	FUNCTION_BLOCK FB 343
	TITLE =G243M COUPLING DEVICE TURNER GERM 8
	//COPYRIGHT:    (C) 2009  BUHLER AG, CH-9240 UZWIL, SWITZERLAND
	//
	//PRODUCT:      WinCoS_BIW01_09
	//
	//TITLE:        COUPLING DEVICE TURNER GERM 8
	//                Machine group control
	//                Maschinengruppensteuerung
	//
	//--------------------------------------------------------------------------------
	//
	//IDENT:        AUTHOR:             DEPT:                              DATE:
	//
	//P01_FB343.1.0 K.Renz              CSB41                              02.Apr.2010
	//             1st Release
	//
	//--------------------------------------------------------------------------------
	//
	//PURPOSE:
	//
	//MANUAL :
	//
	//RESTRICTIONS:
	//
	//--------------------------------------------------------------------------------
	AUTHOR  : KR
	FAMILY  : USW
	VERSION : 9.9


	VAR
	  Gr       : FB10;	//Standard interface to group
	  InOutValue1    : DINT; //Data for user
	  InOutValue2    : DINT; //Data for user
	  OutWayConflict : BOOL;	//Data for user
	  OutSelectionOk : BOOL;	//Data for user
	  CmdNewValue : BOOL;	//Data for user
	  CmdNewJob   : BOOL;	//Data for user
	  OutCodeOK   : BOOL;	//Data for user
	  InEndOfJob  : BOOL ;	//Data for user
	  staWayOk      : BOOL ;	//Data for user
	  EdgeStartRelease : BOOL ;	//Data for user
	  USW8  : BOOL;	//Data for user
	  USW9 : BOOL;	//Data for user
	  USW10: BOOL;	//Data for user
	  USW11: BOOL;	//Data for user
	  USW12: BOOL;	//Data for user
	  USW13: BOOL;	//Data for user
	  USW14: BOOL;	//Data for user
	  USW15: BOOL;	//Data for user
	     #A_2811_MXZ21 : FB12;   // Motor
	     #A_2811_BZS22 : FB14;   // DigInpCont
	     #A_2811_BZS23 : FB14;   // DigInpCont
	     #A_2811_MXZ25 : FB12;   // Motor
	     #A_2811_BZS26 : FB14;   // DigInpCont
	     #A_2811_BZS27 : FB14;   // DigInpCont
	     #A_2811_MXZ31 : FB12;   // Motor
	     #A_2811_BZS32 : FB14;   // DigInpCont
	     #A_2811_BZS33 : FB14;   // DigInpCont
	     #A_2811_MXZ35 : FB12;   // Motor
	     #A_2811_BZS37 : FB14;   // DigInpCont
	     #A_2811_BZS36 : FB14;   // DigInpCont
	END_VAR
	VAR_TEMP
	   tmpEnable		: BOOL;
	   tmpFlag  		: BOOL;
	   tmpCmdNext		: BOOL;
	   tmpLocal  		: BOOL;
	   tmpAspOk  		: BOOL;
	   tmpHWStop 		: BOOL;
	   tmpInstanzDBNo       : INT ;
	END_VAR
	BEGIN
	NETWORK
	TITLE =
	NETWORK
	TITLE =Read command from group control
	//Parameter
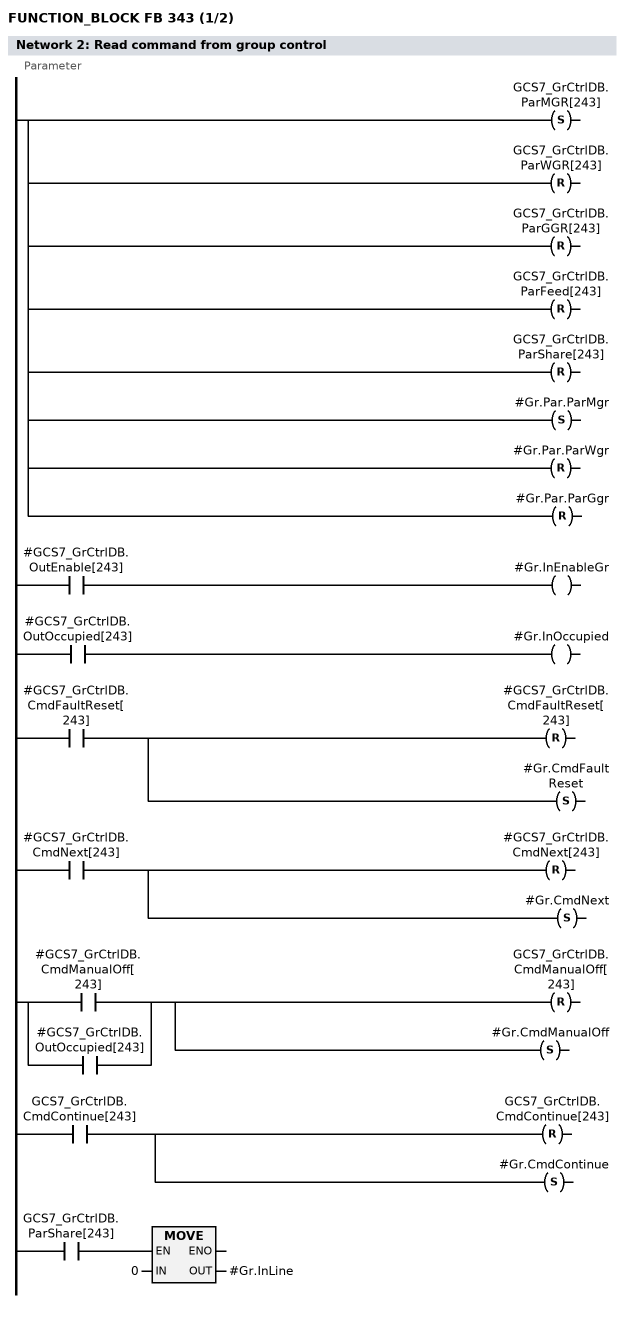
	      SET;
	      S   GCS7_GrCtrlDB.ParMGR[243];
	      R   GCS7_GrCtrlDB.ParWGR[243];
	      R   GCS7_GrCtrlDB.ParGGR[243];
	      R   GCS7_GrCtrlDB.ParFeed[243];
	      R   GCS7_GrCtrlDB.ParShare[243];
	      S   #Gr.Par.ParMgr;
	      R   #Gr.Par.ParWgr;
	      R   #Gr.Par.ParGgr;
	//Command
	      U   #GCS7_GrCtrlDB.OutEnable[243];
	      =   #Gr.InEnableGr;
	      U   #GCS7_GrCtrlDB.OutOccupied[243];
	      =   #Gr.InOccupied;
	      U   #GCS7_GrCtrlDB.CmdFaultReset[243];
	      R   #GCS7_GrCtrlDB.CmdFaultReset[243];
	      S   #Gr.CmdFaultReset;
	      U  #GCS7_GrCtrlDB.CmdNext[243];
	      R   #GCS7_GrCtrlDB.CmdNext[243];
	      S   #Gr.CmdNext;
	      U   #GCS7_GrCtrlDB.CmdManualOff[243];
	      O   #GCS7_GrCtrlDB.OutOccupied[243];
	      R   GCS7_GrCtrlDB.CmdManualOff[243];
	      S   #Gr.CmdManualOff;
	      U  GCS7_GrCtrlDB.CmdContinue[243];
	      R   GCS7_GrCtrlDB.CmdContinue[243];
	      S   #Gr.CmdContinue;
	//Init Line Number
	      U   GCS7_GrCtrlDB.ParShare[243];
	      SPBN WE00;
	      L     0;
	      T     #Gr.InLine;
	WE00: NOP   0;
	NETWORK
	TITLE =Call Methode Control
	// 1. Handle Interface PCControl
	// 2. Prepare mode --> ModePassive,ModeActive,ModeIdling
	// 3. Reset global flags of the group
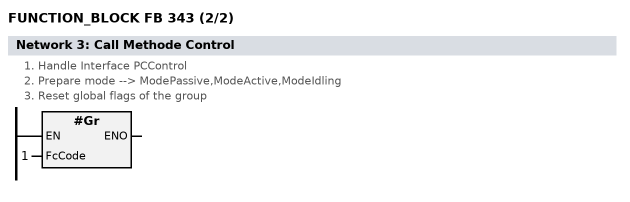
	      CALL #Gr (
	           FcCode                   := 1);
	NETWORK
	TITLE =Restart Idling Time
		L  #Gr.Par.ParIdling;
		L  2;
		>=I;
		SPB IdTm;
		T  #Gr.Par.ParIdling;
	IdTm:   NOP 0;
	      CLR;
	      S    #Gr.CmdRestartIdling;
	NETWORK
	TITLE =Prepare global flags
	NETWORK
	TITLE =Set Pattern (Target position)
	NETWORK
	TITLE =Interlocking WayOk
	//
	NETWORK
	TITLE =Interlocking Autostart
		CLR;
		R   #Gr.OutAutostart;
	NETWORK
	TITLE =Interlocking Enable
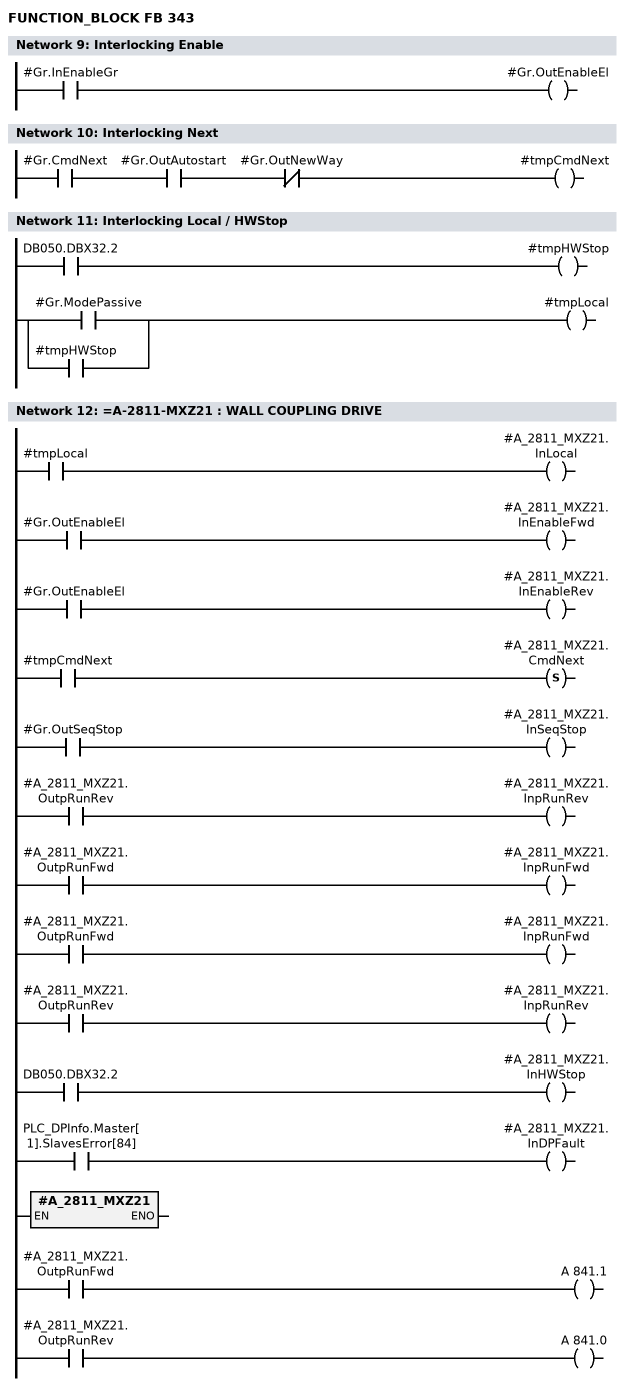
	      U     #Gr.InEnableGr;
	      =     #Gr.OutEnableEl;

	NETWORK
	TITLE =Interlocking Next
	      U     #Gr.CmdNext;
	      U     #Gr.OutAutostart;
	      UN    #Gr.OutNewWay;
	      =    #tmpCmdNext;

	NETWORK
	TITLE =Interlocking Local / HWStop
	      U    DB050.DBX32.2;
	      =    #tmpHWStop;

	      U    #Gr.ModePassive;
	      O    #tmpHWStop;
	      =    #tmpLocal;

	NETWORK
	TITLE ==A-2811-MXZ21 : WALL COUPLING DRIVE
	NOP 0;
	//-InLocal---
	      U     #tmpLocal;
	      =     #A_2811_MXZ21.InLocal;
	//
	//-Interlocking---
	      U     #Gr.OutEnableEl;
	      =     #A_2811_MXZ21.InEnableFwd;
	      U     #Gr.OutEnableEl;
	      =     #A_2811_MXZ21.InEnableRev;
	//
	      U    #tmpCmdNext;
	      S     #A_2811_MXZ21.CmdNext;
	//
	      U     #Gr.OutSeqStop;
	      =     #A_2811_MXZ21.InSeqStop;
	//
	//-Read inputs---
	      U     #A_2811_MXZ21.OutpRunRev;
	      =     #A_2811_MXZ21.InpRunRev;
	      U     #A_2811_MXZ21.OutpRunFwd;
	      =     #A_2811_MXZ21.InpRunFwd;
	      U     #A_2811_MXZ21.OutpRunFwd;
	      =     #A_2811_MXZ21.InpRunFwd;
	      U     #A_2811_MXZ21.OutpRunRev;
	      =     #A_2811_MXZ21.InpRunRev;
	      U   DB050.DBX32.2;
	      =     #A_2811_MXZ21.InHWStop;
	       U     PLC_DPInfo.Master[1].SlavesError[84];
	       =       #A_2811_MXZ21.InDPFault;
	//
	//-Set Parameters---
	//
	//-Call object control---
	      CALL  #A_2811_MXZ21;
	//
	//-Write outputs---
	      U     #A_2811_MXZ21.OutpRunFwd;
	      =     A 841.1;
	      U     #A_2811_MXZ21.OutpRunRev;
	      =     A 841.0;
	NETWORK
	TITLE ==A-2811-BZS22 : COUPLING DRIVE UNLOCKED
	NOP 0;
	//-InLocal---
	      U     #tmpLocal;
	      =     #A_2811_BZS22.InLocal;
	//
	//-Monitoring---
	      CLR;
	      =      #A_2811_BZS22.InMonTrue;
	      CLR;
	      =      #A_2811_BZS22.InMonFalse;
	//
	//-PreAlarm---
	      CLR;
	      =      #A_2811_BZS22.InPreAlarmTrue;
	      CLR;
	      =      #A_2811_BZS22.InPreAlarmFalse;
	//
	//-Additional commands---
	//      CLR
	//      S     #A_2811_BZS22.CmdRunTimeOutTime
	//
	//-Read inputs---
	      U     E 843.0;
	      =     #A_2811_BZS22.InpTrue;
	      U   DB050.DBX32.2;
	      =     #A_2811_BZS22.InHWStop;
	       U     PLC_DPInfo.Master[1].SlavesError[84];
	       =       #A_2811_BZS22.InDPFault;
	//
	//-Set Parameters---
	//
	//-Call object control---
	      CALL  #A_2811_BZS22;
	//
	//-Write outputs---
	NETWORK
	TITLE ==A-2811-BZS23 : COUPLING DRIVE LOCKED
	NOP 0;
	//-InLocal---
	      U     #tmpLocal;
	      =     #A_2811_BZS23.InLocal;
	//
	//-Monitoring---
	      CLR;
	      =      #A_2811_BZS23.InMonTrue;
	      CLR;
	      =      #A_2811_BZS23.InMonFalse;
	//
	//-PreAlarm---
	      CLR;
	      =      #A_2811_BZS23.InPreAlarmTrue;
	      CLR;
	      =      #A_2811_BZS23.InPreAlarmFalse;
	//
	//-Additional commands---
	//      CLR
	//      S     #A_2811_BZS23.CmdRunTimeOutTime
	//
	//-Read inputs---
	      U     E 843.1;
	      =     #A_2811_BZS23.InpTrue;
	      U   DB050.DBX32.2;
	      =     #A_2811_BZS23.InHWStop;
	       U     PLC_DPInfo.Master[1].SlavesError[84];
	       =       #A_2811_BZS23.InDPFault;
	//
	//-Set Parameters---
	//
	//-Call object control---
	      CALL  #A_2811_BZS23;
	//
	//-Write outputs---
	NETWORK
	TITLE ==A-2811-MXZ25 : WALL COUPLING DRIVE
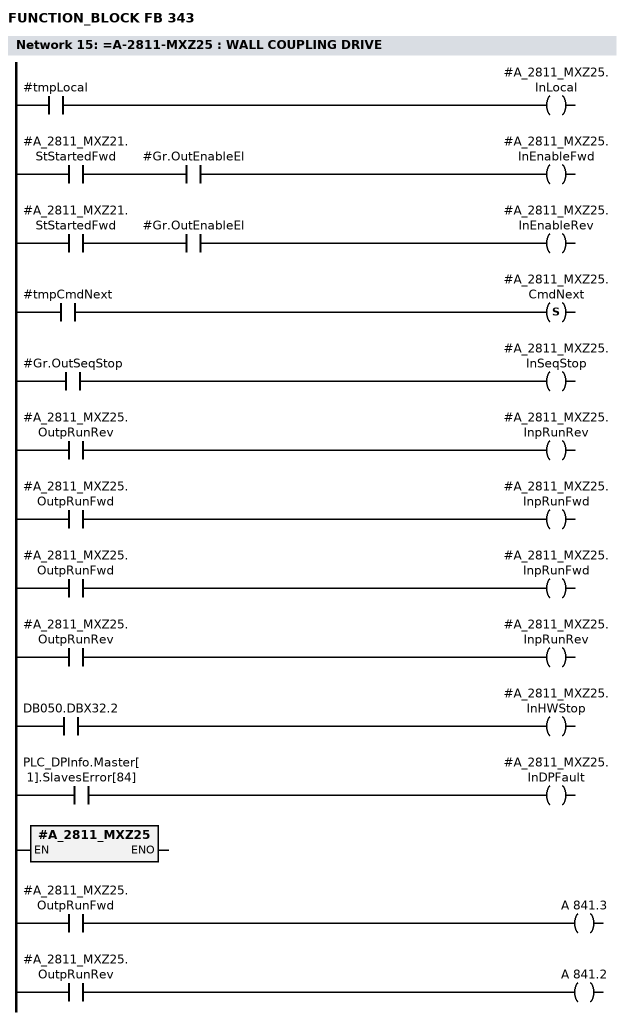
	NOP 0;
	//-InLocal---
	      U     #tmpLocal;
	      =     #A_2811_MXZ25.InLocal;
	//
	//-Interlocking---
	      U     #A_2811_MXZ21.StStartedFwd;
	      U     #Gr.OutEnableEl;
	      =     #A_2811_MXZ25.InEnableFwd;
	      U     #A_2811_MXZ21.StStartedFwd;
	      U     #Gr.OutEnableEl;
	      =     #A_2811_MXZ25.InEnableRev;
	//
	      U    #tmpCmdNext;
	      S     #A_2811_MXZ25.CmdNext;
	//
	      U     #Gr.OutSeqStop;
	      =     #A_2811_MXZ25.InSeqStop;
	//
	//-Read inputs---
	      U     #A_2811_MXZ25.OutpRunRev;
	      =     #A_2811_MXZ25.InpRunRev;
	      U     #A_2811_MXZ25.OutpRunFwd;
	      =     #A_2811_MXZ25.InpRunFwd;
	      U     #A_2811_MXZ25.OutpRunFwd;
	      =     #A_2811_MXZ25.InpRunFwd;
	      U     #A_2811_MXZ25.OutpRunRev;
	      =     #A_2811_MXZ25.InpRunRev;
	      U   DB050.DBX32.2;
	      =     #A_2811_MXZ25.InHWStop;
	       U     PLC_DPInfo.Master[1].SlavesError[84];
	       =       #A_2811_MXZ25.InDPFault;
	//
	//-Set Parameters---
	//
	//-Call object control---
	      CALL  #A_2811_MXZ25;
	//
	//-Write outputs---
	      U     #A_2811_MXZ25.OutpRunFwd;
	      =     A 841.3;
	      U     #A_2811_MXZ25.OutpRunRev;
	      =     A 841.2;
	NETWORK
	TITLE ==A-2811-BZS26 : COUPLING DRIVE UNLOCKED
	NOP 0;
	//-InLocal---
	      U     #tmpLocal;
	      =     #A_2811_BZS26.InLocal;
	//
	//-Monitoring---
	      CLR;
	      =      #A_2811_BZS26.InMonTrue;
	      CLR;
	      =      #A_2811_BZS26.InMonFalse;
	//
	//-PreAlarm---
	      CLR;
	      =      #A_2811_BZS26.InPreAlarmTrue;
	      CLR;
	      =      #A_2811_BZS26.InPreAlarmFalse;
	//
	//-Additional commands---
	//      CLR
	//      S     #A_2811_BZS26.CmdRunTimeOutTime
	//
	//-Read inputs---
	      U     E 843.2;
	      =     #A_2811_BZS26.InpTrue;
	      U   DB050.DBX32.2;
	      =     #A_2811_BZS26.InHWStop;
	       U     PLC_DPInfo.Master[1].SlavesError[84];
	       =       #A_2811_BZS26.InDPFault;
	//
	//-Set Parameters---
	//
	//-Call object control---
	      CALL  #A_2811_BZS26;
	//
	//-Write outputs---
	NETWORK
	TITLE ==A-2811-BZS27 : COUPLING DRIVE LOCKED
	NOP 0;
	//-InLocal---
	      U     #tmpLocal;
	      =     #A_2811_BZS27.InLocal;
	//
	//-Monitoring---
	      CLR;
	      =      #A_2811_BZS27.InMonTrue;
	      CLR;
	      =      #A_2811_BZS27.InMonFalse;
	//
	//-PreAlarm---
	      CLR;
	      =      #A_2811_BZS27.InPreAlarmTrue;
	      CLR;
	      =      #A_2811_BZS27.InPreAlarmFalse;
	//
	//-Additional commands---
	//      CLR
	//      S     #A_2811_BZS27.CmdRunTimeOutTime
	//
	//-Read inputs---
	      U     E 843.3;
	      =     #A_2811_BZS27.InpTrue;
	      U   DB050.DBX32.2;
	      =     #A_2811_BZS27.InHWStop;
	       U     PLC_DPInfo.Master[1].SlavesError[84];
	       =       #A_2811_BZS27.InDPFault;
	//
	//-Set Parameters---
	//
	//-Call object control---
	      CALL  #A_2811_BZS27;
	//
	//-Write outputs---
	NETWORK
	TITLE ==A-2811-MXZ31 : WALL COUPLING DRIVE
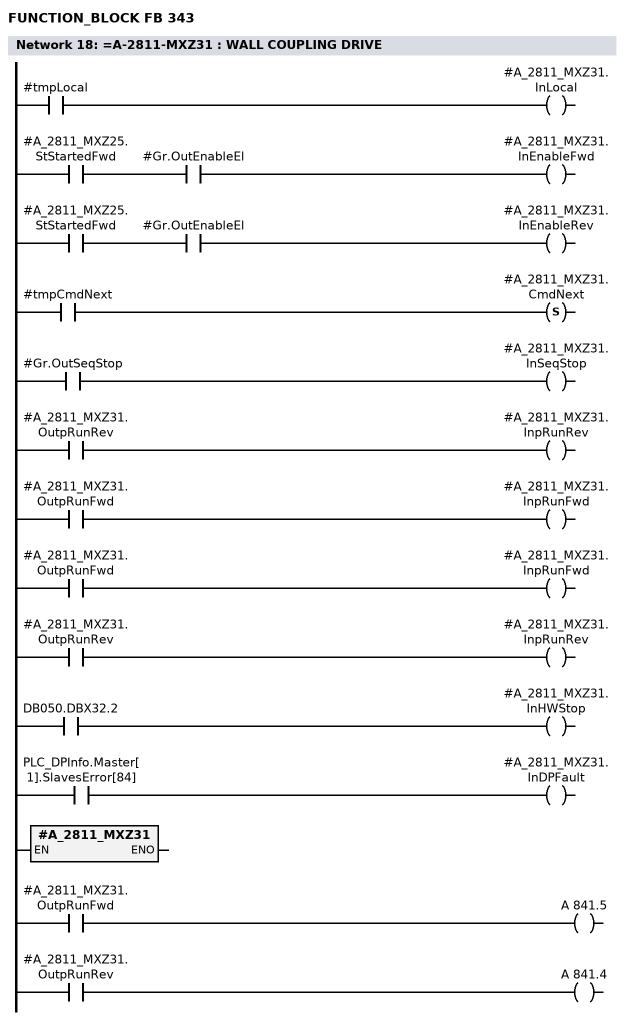
	NOP 0;
	//-InLocal---
	      U     #tmpLocal;
	      =     #A_2811_MXZ31.InLocal;
	//
	//-Interlocking---
	      U     #A_2811_MXZ25.StStartedFwd;
	      U     #Gr.OutEnableEl;
	      =     #A_2811_MXZ31.InEnableFwd;
	      U     #A_2811_MXZ25.StStartedFwd;
	      U     #Gr.OutEnableEl;
	      =     #A_2811_MXZ31.InEnableRev;
	//
	      U    #tmpCmdNext;
	      S     #A_2811_MXZ31.CmdNext;
	//
	      U     #Gr.OutSeqStop;
	      =     #A_2811_MXZ31.InSeqStop;
	//
	//-Read inputs---
	      U     #A_2811_MXZ31.OutpRunRev;
	      =     #A_2811_MXZ31.InpRunRev;
	      U     #A_2811_MXZ31.OutpRunFwd;
	      =     #A_2811_MXZ31.InpRunFwd;
	      U     #A_2811_MXZ31.OutpRunFwd;
	      =     #A_2811_MXZ31.InpRunFwd;
	      U     #A_2811_MXZ31.OutpRunRev;
	      =     #A_2811_MXZ31.InpRunRev;
	      U   DB050.DBX32.2;
	      =     #A_2811_MXZ31.InHWStop;
	       U     PLC_DPInfo.Master[1].SlavesError[84];
	       =       #A_2811_MXZ31.InDPFault;
	//
	//-Set Parameters---
	//
	//-Call object control---
	      CALL  #A_2811_MXZ31;
	//
	//-Write outputs---
	      U     #A_2811_MXZ31.OutpRunFwd;
	      =     A 841.5;
	      U     #A_2811_MXZ31.OutpRunRev;
	      =     A 841.4;
	NETWORK
	TITLE ==A-2811-BZS32 : COUPLING DRIVE UNLOCKED
	NOP 0;
	//-InLocal---
	      U     #tmpLocal;
	      =     #A_2811_BZS32.InLocal;
	//
	//-Monitoring---
	      CLR;
	      =      #A_2811_BZS32.InMonTrue;
	      CLR;
	      =      #A_2811_BZS32.InMonFalse;
	//
	//-PreAlarm---
	      CLR;
	      =      #A_2811_BZS32.InPreAlarmTrue;
	      CLR;
	      =      #A_2811_BZS32.InPreAlarmFalse;
	//
	//-Additional commands---
	//      CLR
	//      S     #A_2811_BZS32.CmdRunTimeOutTime
	//
	//-Read inputs---
	      U     E 843.4;
	      =     #A_2811_BZS32.InpTrue;
	      U   DB050.DBX32.2;
	      =     #A_2811_BZS32.InHWStop;
	       U     PLC_DPInfo.Master[1].SlavesError[84];
	       =       #A_2811_BZS32.InDPFault;
	//
	//-Set Parameters---
	//
	//-Call object control---
	      CALL  #A_2811_BZS32;
	//
	//-Write outputs---
	NETWORK
	TITLE ==A-2811-BZS33 : COUPLING DRIVE LOCKED
	NOP 0;
	//-InLocal---
	      U     #tmpLocal;
	      =     #A_2811_BZS33.InLocal;
	//
	//-Monitoring---
	      CLR;
	      =      #A_2811_BZS33.InMonTrue;
	      CLR;
	      =      #A_2811_BZS33.InMonFalse;
	//
	//-PreAlarm---
	      CLR;
	      =      #A_2811_BZS33.InPreAlarmTrue;
	      CLR;
	      =      #A_2811_BZS33.InPreAlarmFalse;
	//
	//-Additional commands---
	//      CLR
	//      S     #A_2811_BZS33.CmdRunTimeOutTime
	//
	//-Read inputs---
	      U     E 843.5;
	      =     #A_2811_BZS33.InpTrue;
	      U   DB050.DBX32.2;
	      =     #A_2811_BZS33.InHWStop;
	       U     PLC_DPInfo.Master[1].SlavesError[84];
	       =       #A_2811_BZS33.InDPFault;
	//
	//-Set Parameters---
	//
	//-Call object control---
	      CALL  #A_2811_BZS33;
	//
	//-Write outputs---
	NETWORK
	TITLE ==A-2811-MXZ35 : WALL COUPLING DRIVE
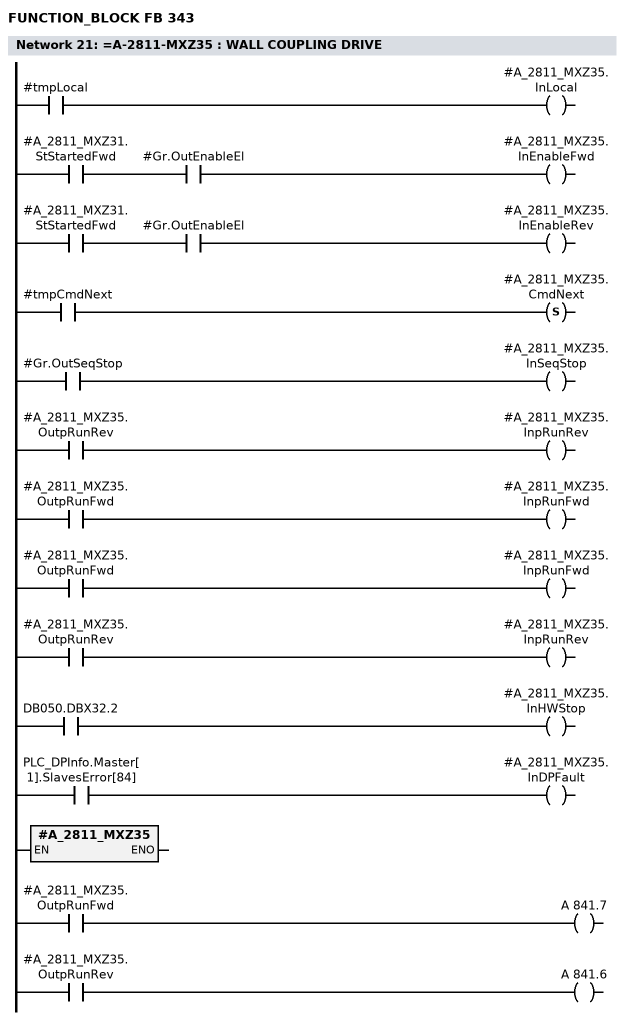
	NOP 0;
	//-InLocal---
	      U     #tmpLocal;
	      =     #A_2811_MXZ35.InLocal;
	//
	//-Interlocking---
	      U     #A_2811_MXZ31.StStartedFwd;
	      U     #Gr.OutEnableEl;
	      =     #A_2811_MXZ35.InEnableFwd;
	      U     #A_2811_MXZ31.StStartedFwd;
	      U     #Gr.OutEnableEl;
	      =     #A_2811_MXZ35.InEnableRev;
	//
	      U    #tmpCmdNext;
	      S     #A_2811_MXZ35.CmdNext;
	//
	      U     #Gr.OutSeqStop;
	      =     #A_2811_MXZ35.InSeqStop;
	//
	//-Read inputs---
	      U     #A_2811_MXZ35.OutpRunRev;
	      =     #A_2811_MXZ35.InpRunRev;
	      U     #A_2811_MXZ35.OutpRunFwd;
	      =     #A_2811_MXZ35.InpRunFwd;
	      U     #A_2811_MXZ35.OutpRunFwd;
	      =     #A_2811_MXZ35.InpRunFwd;
	      U     #A_2811_MXZ35.OutpRunRev;
	      =     #A_2811_MXZ35.InpRunRev;
	      U   DB050.DBX32.2;
	      =     #A_2811_MXZ35.InHWStop;
	       U     PLC_DPInfo.Master[1].SlavesError[84];
	       =       #A_2811_MXZ35.InDPFault;
	//
	//-Set Parameters---
	//
	//-Call object control---
	      CALL  #A_2811_MXZ35;
	//
	//-Write outputs---
	      U     #A_2811_MXZ35.OutpRunFwd;
	      =     A 841.7;
	      U     #A_2811_MXZ35.OutpRunRev;
	      =     A 841.6;
	NETWORK
	TITLE ==A-2811-BZS36 : COUPLING DRIVE UNLOCKED
	NOP 0;
	//-InLocal---
	      U     #tmpLocal;
	      =     #A_2811_BZS36.InLocal;
	//
	//-Monitoring---
	      CLR;
	      =      #A_2811_BZS36.InMonTrue;
	      CLR;
	      =      #A_2811_BZS36.InMonFalse;
	//
	//-PreAlarm---
	      CLR;
	      =      #A_2811_BZS36.InPreAlarmTrue;
	      CLR;
	      =      #A_2811_BZS36.InPreAlarmFalse;
	//
	//-Additional commands---
	//      CLR
	//      S     #A_2811_BZS36.CmdRunTimeOutTime
	//
	//-Read inputs---
	      U     E 843.6;
	      =     #A_2811_BZS36.InpTrue;
	      U   DB050.DBX32.2;
	      =     #A_2811_BZS36.InHWStop;
	       U     PLC_DPInfo.Master[1].SlavesError[84];
	       =       #A_2811_BZS36.InDPFault;
	//
	//-Set Parameters---
	//
	//-Call object control---
	      CALL  #A_2811_BZS36;
	//
	//-Write outputs---
	NETWORK
	TITLE ==A-2811-BZS37 : COUPLING DRIVE LOCKED
	NOP 0;
	//-InLocal---
	      U     #tmpLocal;
	      =     #A_2811_BZS37.InLocal;
	//
	//-Monitoring---
	      CLR;
	      =      #A_2811_BZS37.InMonTrue;
	      CLR;
	      =      #A_2811_BZS37.InMonFalse;
	//
	//-PreAlarm---
	      CLR;
	      =      #A_2811_BZS37.InPreAlarmTrue;
	      CLR;
	      =      #A_2811_BZS37.InPreAlarmFalse;
	//
	//-Additional commands---
	//      CLR
	//      S     #A_2811_BZS37.CmdRunTimeOutTime
	//
	//-Read inputs---
	      U     E 843.7;
	      =     #A_2811_BZS37.InpTrue;
	      U   DB050.DBX32.2;
	      =     #A_2811_BZS37.InHWStop;
	       U     PLC_DPInfo.Master[1].SlavesError[84];
	       =       #A_2811_BZS37.InDPFault;
	//
	//-Set Parameters---
	//
	//-Call object control---
	      CALL  #A_2811_BZS37;
	//
	//-Write outputs---
	NETWORK
	TITLE =Test Fault
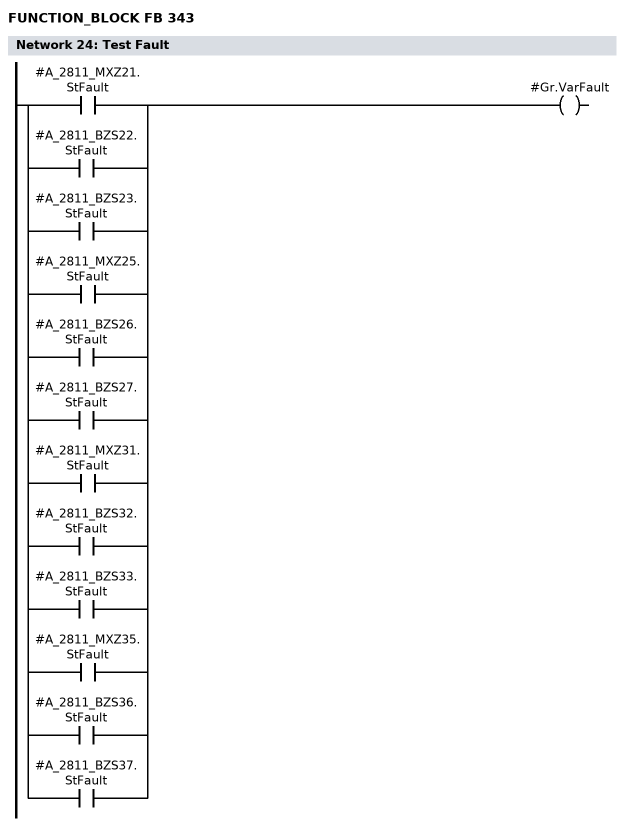
	      U     #A_2811_MXZ21.StFault;
	      O     #A_2811_BZS22.StFault;
	      O     #A_2811_BZS23.StFault;
	      O     #A_2811_MXZ25.StFault;
	      O     #A_2811_BZS26.StFault;
	      O     #A_2811_BZS27.StFault;
	      O     #A_2811_MXZ31.StFault;
	      O     #A_2811_BZS32.StFault;
	      O     #A_2811_BZS33.StFault;
	      O     #A_2811_MXZ35.StFault;
	      O     #A_2811_BZS36.StFault;
	      O     #A_2811_BZS37.StFault;
	      =     #Gr.VarFault;
	NETWORK
	TITLE =Test Warning
	      CLR;
	      =     #Gr.OutWarning;
	NETWORK
	TITLE =Test Stopped
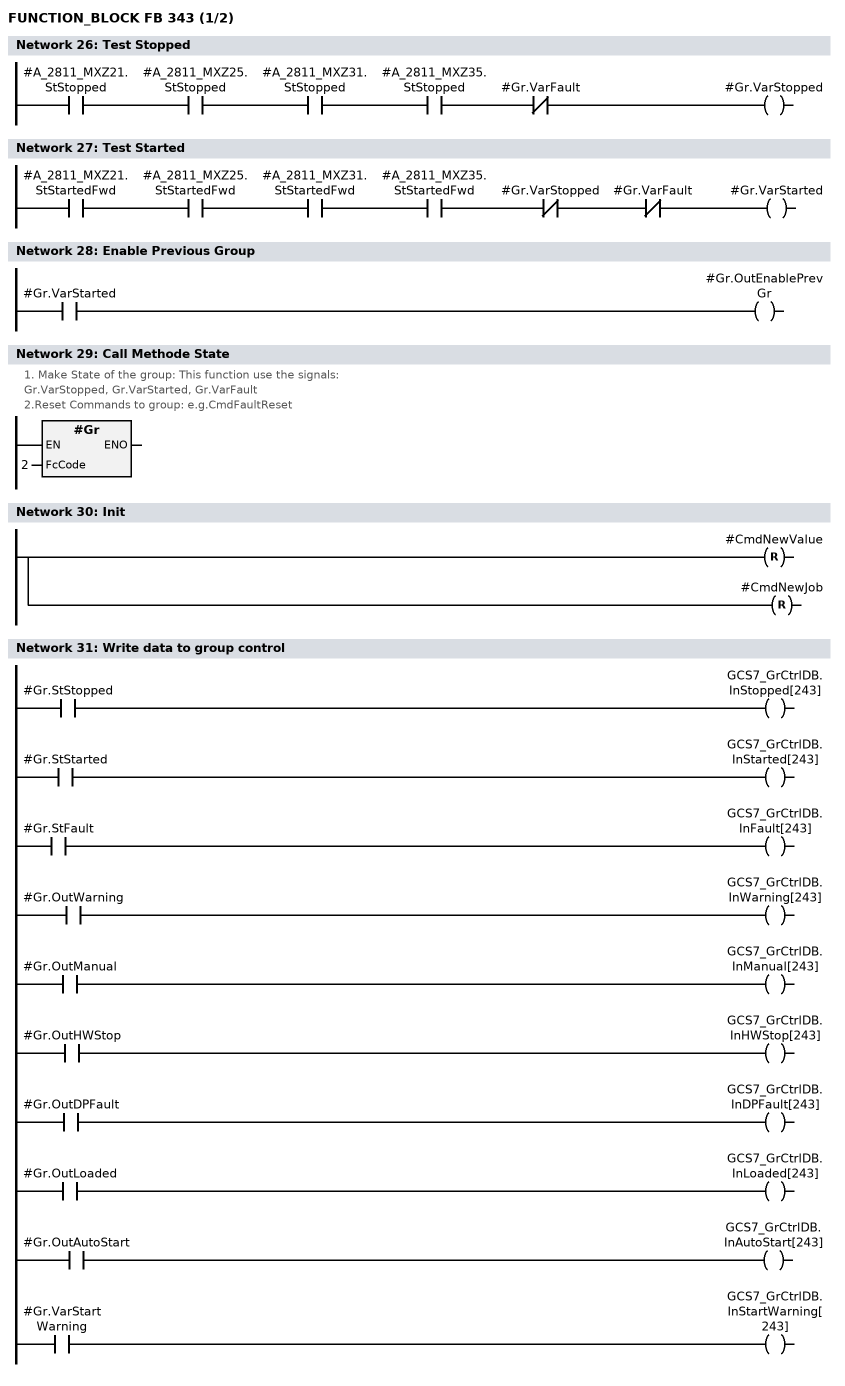
	      U     #A_2811_MXZ21.StStopped;
	      U     #A_2811_MXZ25.StStopped;
	      U     #A_2811_MXZ31.StStopped;
	      U     #A_2811_MXZ35.StStopped;
	      UN   #Gr.VarFault;
	      =     #Gr.VarStopped;
	NETWORK
	TITLE =Test Started
	      U     #A_2811_MXZ21.StStartedFwd;
	      U     #A_2811_MXZ25.StStartedFwd;
	      U     #A_2811_MXZ31.StStartedFwd;
	      U     #A_2811_MXZ35.StStartedFwd;
	      UN  #Gr.VarStopped;
	      UN  #Gr.VarFault;
	      =     #Gr.VarStarted;
	NETWORK
	TITLE =Enable Previous Group
	      U    #Gr.VarStarted;
	      =     #Gr.OutEnablePrevGr;
	NETWORK
	TITLE =Call Methode State
	//1. Make State of the group: This function use the signals:
	//        Gr.VarStopped, Gr.VarStarted, Gr.VarFault
	//2.Reset Commands to group: e.g.CmdFaultReset
	      CALL #Gr (
	           FcCode                   := 2);
	NETWORK
	TITLE =Init
	      SET;
	      R    #CmdNewValue;
	      R    #CmdNewJob;
	NETWORK
	TITLE =Write data to group control
	      U   #Gr.StStopped;
	      =   GCS7_GrCtrlDB.InStopped[243];
	      U   #Gr.StStarted;
	      =   GCS7_GrCtrlDB.InStarted[243];
	      U   #Gr.StFault;
	      =   GCS7_GrCtrlDB.InFault[243];
	      U   #Gr.OutWarning;
	      =   GCS7_GrCtrlDB.InWarning[243];
	      U   #Gr.OutManual;
	      =   GCS7_GrCtrlDB.InManual[243];
	      U   #Gr.OutHWStop;
	      =   GCS7_GrCtrlDB.InHWStop[243];
	      U   #Gr.OutDPFault;
	      =   GCS7_GrCtrlDB.InDPFault[243];
	      U   #Gr.OutLoaded;
	      =   GCS7_GrCtrlDB.InLoaded[243];
	      U   #Gr.OutAutoStart;
	      =   GCS7_GrCtrlDB.InAutoStart[243];
	      U   #Gr.VarStartWarning;
	      =   GCS7_GrCtrlDB.InStartWarning[243];
	NETWORK
	TITLE =End of block
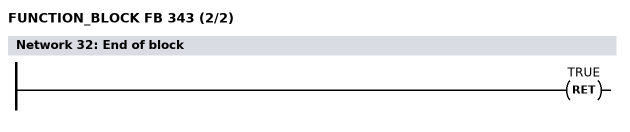

	BE

	END_FUNCTION_BLOCK
